FUNCTION IntegerLesen : INT
VAR_INPUT
	LowByte: BYTE;
	HighByte: BYTE;
END_VAR
VAR
	DoppelByte: WORD;
END_VAR

DoppelByte := 256 * LowByte + HighByte;	// Siemens fährt ja Little Endian
IntegerLesen := WORD_TO_INT(DoppelByte);

END_FUNCTION

(* stored: Version 1.1.0.1, ProductVersion 3.1.4024.5
   POU IntegerLesen: Id {a6a4413c-8c3c-42d0-b546-1186666f9e91}, SpecialFunc None *)
